Staubli VAL3: GenericConv.pjx

--- GenericConv.pjx ---
Parameters version=s7.3 stackSize=5000 millimeterUnit=true
Program file=checkTrackArea.pgx
Program file=conveyor.pgx
Program file=create.pgx
Program file=disableQueue.pgx
Program file=enableQueue.pgx
Program file=fillQueue.pgx
Program file=flushQueue.pgx
Program file=getConvFrame.pgx
Program file=getDetectDist.pgx
Program file=getDetectFrame.pgx
Program file=getDistance.pgx
Program file=getErrorMessage.pgx
Program file=getNextID.pgx
Program file=getObjectData.pgx
Program file=getObjectLatch.pgx
Program file=getObjectOffset.pgx
Program file=getObjectPos.pgx
Program file=getStatus.pgx
Program file=getTravelDist.pgx
Program file=init.pgx
Program file=kill.pgx
Program file=releaseObject.pgx
Program file=removePart.pgx
Program file=reset.pgx
Program file=setCalibrating.pgx
Program file=setConveyor.pgx
Program file=setObjectInUse.pgx
Program file=start.pgx
Program file=stop.pgx
Program file=teach.pgx
Program file=whichObjectUsed.pgx
Data file=GenericConv.dtx
Library alias=cfg path=Disk://Tracking/config/config.pjx
Library alias=det path=Disk://Tracking/Templates/GenericDetect/GenericDetect.pjx autoload=false
Library alias=enc path=Disk://Tracking/Templates/GenericEnc/GenericEnc.pjx autoload=false
Library alias=geometry path=Disk://Tracking/Templates/Geometry/Geometry.pjx autoload=false
Library alias=swap path=Disk://Tracking/Swap/Swap.pjx
Library alias=ut path=Disk://Tracking/Tools/util/util.pjx
Library alias=lang path=Disk://Tracking/language/english/english.pjx
Library alias=out path=Disk://Tracking/io/outputs/outputs.pjx

--- getDetectFrame.pgx ---
public program getDetectFrame(frame& x_fDetection, frame x_fRefFrame, num& x_nError)
  local string l_sCustomTxt[2]
begin
  // This program returns the position of the conveyor frame
  // in the réference frame passed as parameter
  //
  // Input param
  //  x_fRefFrame   : Reference frame in which the position of the conveyor
  //                frame must be returned
  //
  // Output param
  //  x_fConveyor   : Conveyor frame
  //  x_nError      : Error code
  //    0    --> No error
  //    14   --> Conveyor library not started, the frame cannot be computed.
  //
  // Created 7-03-08                                   C.CURRIVAND
  //----------------------------------------------------------------
  x_nError=0
  if bInit
    x_fDetection.trsf=position(fDetection,x_fRefFrame)
  else
    x_nError=14
    // Prepare clear text error message
    l_sCustomTxt[0]=sConveyorName
    l_sCustomTxt[1]="detection"
    call ut:addStrToString(lang:sListOfMessage[x_nError],sErrorMessage,"",l_sCustomTxt)
  endIf
end

--- init.pgx ---
public program init(num x_nConvNum, num& x_nError)
  local num l_i
  local bool l_bSigClockOk
  local bool l_bQuit
  local trsf l_tfCenter
  local trsf l_tfConveyor
  local num l_nError
  local num l_nStep
  local string l_sFileToLoad
  local trsf l_TRSF
begin
  // This program initializes the conveyor library
  //
  // Input param
  //  x_nConvNum : Conveyor number
  //
  // Output param
  //  x_nError : Error code
  //        =0 : No error
  //        =33: Error while loading geometry library
  //        =31: Error while loading encoder library
  //        =32: Error while loading detection library
  //
  //----------------------------------------------------------------
  //
  //
  bInit=false
  l_bQuit=false
  x_nError=0
  nStatus=0
  sConvNum="CNV"+toString("",x_nConvNum)
  //***************************
  //*****   Constant values ***
  //***************************
  nSysCycleTime=sel(left(getVersion("ArmType"),2)=="tp",0.002,0.004)
  nFirDelay=nSysCycleTime*2
  nFirTime=nSysCycleTime*nFirOrdre
  nPUSH_NEGATIVE=10
  nDETECT_OVR=11
  //***************************
  //*****   Libraries   *******
  //***************************
  do
    switch l_nStep
      // --- Load Geometry library
      case 0
        l_sFileToLoad=cfg:sPATHCONVEYOR+sConveyorName+"\"+sGeometryLib
        l_nError=geometry:libLoad(l_sFileToLoad)
        if l_nError!=0
          x_nError=33
          if bAnd(cfg:nLog,cfg:nLOGMISC)==cfg:nLOGMISC
            ? sConvNum+"(init)>>Loading geometry library "+l_sFileToLoad+", status "+toString("0",l_nError)
          endIf
          l_bQuit=true
        else
          l_nStep=10
        endIf
      break
      // --- Load Encoder library
      case 10
        l_sFileToLoad=cfg:sPATHENCODER+sEncoderLib
        l_nError=enc:libLoad(l_sFileToLoad)
        if l_nError!=0
          x_nError=31
          if bAnd(cfg:nLog,cfg:nLOGMISC)==cfg:nLOGMISC
            ? sConvNum+"(init)>>Loading encoder library "+l_sFileToLoad+", status:"+toString("0",l_nError)
          endIf
          l_bQuit=true
        else
          l_nStep=20
        endIf
      break
      // --- Load Detection library
      case 20
        l_sFileToLoad=cfg:sPATHDETECTION+sDetectionLib
        l_nError=det:libLoad(l_sFileToLoad)
        if l_nError!=0
          x_nError=32
          if bAnd(cfg:nLog,cfg:nLOGMISC)==cfg:nLOGMISC
            ? sConvNum+"(init)>>Loading detection library "+l_sFileToLoad+", status:"+toString("0",l_nError)
          endIf
        endIf
        l_bQuit=true
      break
    endSwitch
    delay(0)
  until (l_bQuit==true)
  //
  // If error while loading libraries, prepare clear text
  // else continue with initialisations
  if x_nError!=0
    // Prepare clear text error message
    call ut:addStrToString(lang:sListOfMessage[x_nError],sErrorMessage,"",l_sFileToLoad)
    call ut:addNumToString(sErrorMessage,sErrorMessage,"*",l_nError)
  else
    //******************************
    //*****  Tracking Queues  ******
    //******************************
    // --- Resize arrays according to nBufferSize
    resize(nEncLatchedVal,1,nBufferSize)
    resize(nQueueID,1,nBufferSize)
    resize(nNumbOfUser,1,nBufferSize)
    resize(trDetectedCoord,1,nBufferSize)
    //
    // -- Resize temporarily buffers
    resize(nTmpID,1,det:nMaxNumOfObject)
    resize(nTmpEncLatched,1,det:nMaxNumOfObject)
    resize(trTmp,1,det:nMaxNumOfObject)
    //
    // --- Initialize tracking queues
    for l_i=0 to (nBufferSize-1)
      nEncLatchedVal[l_i]=0
      trDetectedCoord[l_i]=trDEFAULT
      nQueueID[l_i]=nDEFAULTID
      nNumbOfUser[l_i]=0
    endFor
    //
    //***************************
    //*****   Locations    ******
    //***************************
    //
    call geometry:GetPoint(1)
    //
    //***************************
    //*****   Frames       ******
    //***************************
    call geometry:BuildFrame("conveyor",fConveyor,l_nError)
    if l_nError!=0
      logMsg(sConvNum+"(init)>>Cannot compute conveyor frame : "+toString("0",l_nError))
    endIf
    call geometry:BuildFrame("vision",fDetection,l_nError)
    if l_nError!=0
      logMsg(sConvNum+"(init)>>Warning,cannot compute vision frame : "+toString("0",l_nError))
    endIf
    //
    if bUseUserCenter
      l_tfConveyor=fConveyor.trsf
      l_tfCenter=swap:trWinCenter
      l_tfConveyor.x=l_tfCenter.x
      l_tfConveyor.y=l_tfCenter.y
      l_tfConveyor.z=l_tfCenter.z
      fConveyor.trsf=l_tfConveyor
    endIf
    //***************************
    //***** Digital output ******
    //***************************
    // The conveyor library is able to deliver a clock signal depending on
    // the advance of the conveyor .
    //-- Clock signal to trigger detection device
    l_nError = getData("out:"+sClockSigName,doClock)
    l_bSigClockOk=(ioStatus(doClock)>=0) and l_nError != -1
    //
    //***************************
    //*****   Booleans     ******
    //***************************
    //
    det:bTaskDetOK=false
    bInit=true
    bResetConv=false
    //
    bLinear=geometry:bLinear
    // Mutex boolean for accessing the object queue
    bLockQueueAcces=false
    //--- Evaluate if clock feature is enabled
    bClockEnabled=(nClockPeriod>0) and (l_bSigClockOk==true)
    //
    //Enable queuing of the detected objects
    call enableQueue()
    //
    //***************************
    //*****   Numerics     ******
    //***************************
    //
    nIdxPush=0
    nIdxPull=0
    nAddedToQueue=0
    //--- Select robot's working area boundaries
    if bLinear
      trBoundaryUp[0]=!fConveyor.trsf*swap:trWinUp[0]
      trBoundaryUp[1]=!fConveyor.trsf*swap:trWinUp[1]
      trBoundaryDwn[0]=!fConveyor.trsf*swap:trWinDown[0]
      trBoundaryDwn[1]=!fConveyor.trsf*swap:trWinDown[1]
      // Make volume a trapezoidal shape. Alternatively compute equation of the edge (more complex)
      trBoundaryDwn[0].y=trBoundaryUp[0].y
      trBoundaryDwn[1].y=trBoundaryUp[1].y
      //
      // Compute equation of upstream boundary in conveyor frame
      if abs((trBoundaryUp[1].x-trBoundaryUp[0].x))>0.001
        nA1=(trBoundaryUp[1].y-trBoundaryUp[0].y)/(trBoundaryUp[1].x-trBoundaryUp[0].x)
      else
        nA1=0
      endIf
      nB1=-nA1*trBoundaryUp[0].x
      // Compute equation of downstream boundary in conveyor frame
      if abs((trBoundaryDwn[1].x-trBoundaryDwn[0].x))>0.001
        nA2=(trBoundaryDwn[1].y-trBoundaryDwn[0].y)/(trBoundaryDwn[1].x-trBoundaryDwn[0].x)
      else
        nA2=0
      endIf
      nB2=-nA2*trBoundaryDwn[0].x
    else
      l_TRSF=!fConveyor.trsf*swap:trWinDown[0]
      nBoundaryDwn=atan(l_TRSF.y/l_TRSF.x)
      l_TRSF=!fConveyor.trsf*swap:trWinUp[0]
      nBoundaryUp=atan(l_TRSF.y/l_TRSF.x)
    endIf
    // Override limits with user limits
    if bUseUserLimit==true
      //      trBoundaryDwn={nWinDownStream,0,0,0,0,0}
      //      trBoundaryUp={nWinUpStream,0,0,0,0,0}
    endIf
    //
  endIf
  //
end

--- releaseObject.pgx ---
public program releaseObject(num x_nIdx)
  local string l_str
  local num l_nQueue
  local string l_sMessage
begin
  // This programs is used to count how many users have accessed
  // to the data of an object in the queue
  //
  // Input param
  //  x_nIdx       : Index of the object in the queue
  //
  // Output param
  //  none
  //
  // Created 25-09-07                                   C.CURRIVAND
  //----------------------------------------------------------------
  //
  nNumbOfUser[x_nIdx]=max(0,nNumbOfUser[x_nIdx]-1)
  if (roundDown(nNumbOfUser[x_nIdx])<=0)
    nQueueID[x_nIdx]=-1
    //
    if bAnd(cfg:nLog,cfg:nLOGQUEUE)==cfg:nLOGQUEUE
      ? sConvNum+"(releaseObject)>>"
      ? "           -------------------------Remove Part------------------------"
      ? "           |Index|  ID | latch value |     x    |     y    |    rz    |"
      ? "           ------------------------------------------------------------"
      for l_nQueue=0 to nBufferSize-1
        if nQueueID[l_nQueue]>=0
          l_sMessage="           | "+toString("3.0",l_nQueue)+" | "+toString("3.0",nQueueID[l_nQueue])+" | "+toString("11.2",nEncLatchedVal[l_nQueue])+" | "
          l_sMessage=l_sMessage+toString("8.2",trDetectedCoord[l_nQueue].x)+" | "+toString("8.2",trDetectedCoord[l_nQueue].y)+" | "+toString("8.2",trDetectedCoord[l_nQueue].rz)+" |"
          ? l_sMessage
        endIf
      endFor
      ? "           ------------------------------------------------------------"
      ? ""
    endIf
    //
  endIf
  if bAnd(cfg:nLog,cfg:nLOGMOTION)==cfg:nLOGMOTION
    l_str=sConvNum+"(releaseObject)>>Request to release object @ position "+toString("",x_nIdx)+" in queue, nbUser="
    l_str=l_str+toString("",nNumbOfUser[x_nIdx])
    ? l_str
  endIf
end

--- removePart.pgx ---
public program removePart()
begin
  setMutex(bLockQueueAcces)
  //
  if bAnd(cfg:nLog,cfg:nLOGMOTION)==cfg:nLOGMOTION
    ? sConvNum+"(removePart)>>Request to remove object @ position "+toString("",nIdxPull)+" Push: "+toString("",nIdxPush)
  endIf
  //
  if nIdxPull!=nIdxPush
    call releaseObject(nIdxPull)
    nIdxPull=(nIdxPull+1)%nBufferSize
  endIf
  //
  bLockQueueAcces=false
end
